// TIA Portal V17 export
// export: Created 2022-07-20T07:02:30.5184204Z, ExportSetting WithDefaults, DisplayName Totally Integrated Automation Portal, DisplayVersion V17, DisplayName TIA Portal Openness, DisplayVersion V17, DisplayName TIA Portal Version Control Interface, DisplayVersion V17, DisplayName SINAMICS Startdrive Advanced, DisplayVersion V17, DisplayName SINAMICS Startdrive G130, G150, S120, S150, SINAMICS MV, S210, DisplayVersion V17, DisplayName SINAMICS Startdrive G110M, G120, G120C, G120D, G120P, G115D, DisplayVersion V17, DisplayName STEP 7 Professional, DisplayVersion V17, DisplayName STEP 7 Safety, DisplayVersion V17, DisplayName WinCC Advanced, DisplayVersion V17
FUNCTION_BLOCK "FB11003_CamConvertProfile"   // FB11003, LAD
TITLE = Transfert and check data of foil profile
{ S7_Optimized_Access := 'TRUE' }
VERSION : 0.1
// stored: AutoNumber false, IsIECCheckEnabled false, IsRetainMemResEnabled false, MemoryReserve 100, SetENOAutomatically false, UDAEnableTagReadback false
   VAR_INPUT
      SheetProfile { ExternalAccessible := 'False'; ExternalVisible := 'False'; ExternalWritable := 'False'} : "stSheetProfile";
      FoilAcceleration : Real;
      FoilDeceleration : Real;
      RatioFoilPaper : Real := 1.0;
      CompensationForTensionInAcceleration : Real;
      CompensationForTensionInDeceleration : Real;
      MainDriveVelocity : Real;
      DistanceProductSensorFilmDrum : Real;
      Execute { ExternalAccessible := 'False'; ExternalVisible := 'False'; ExternalWritable := 'False'} : Bool;
   END_VAR
   VAR_OUTPUT
      Done { ExternalAccessible := 'False'; ExternalVisible := 'False'; ExternalWritable := 'False'} : Bool;
      Error { ExternalAccessible := 'False'; ExternalVisible := 'False'; ExternalWritable := 'False'} : Bool;
      DeadZoneBeforeStampArea { ExternalAccessible := 'False'; ExternalVisible := 'False'; ExternalWritable := 'False'} : Real;
      DeadZoneAfterStampArea { ExternalAccessible := 'False'; ExternalVisible := 'False'; ExternalWritable := 'False'} : Real;
      GapBetweenArea : Real;
      NbPoints : Real;
      CamProfile { ExternalAccessible := 'False'; ExternalVisible := 'False'; ExternalWritable := 'False'} : Array[1..32] of "LCamHdl_typeBasicPoint";
   END_VAR
   VAR
      statNumberOfArea : UInt;
      FoilAccelerationDistance : Real;   // [mm]
      FoilDecelerationDistance : Real;   // [mm]
      MasterAccelerationDistance : Real;
      MasterDecelerationDistance : Real;
      statPointtNumber { ExternalAccessible := 'False'; ExternalVisible := 'False'; ExternalWritable := 'False'} : UInt;
      statDone : Bool;
      statError : Bool;
      R_TRIG_Execute : R_TRIG;
   END_VAR
   VAR_TEMP
      AreaNumber : UInt;
      tempTotLength : Real;
   END_VAR
   VAR CONSTANT
      ratioDeadZone : Real := 4.0;
   END_VAR
   // // SheetProfile.Length : [mm]
BEGIN

REGION Network 1 (SCL): Comments
   //==========================================================================================
   // SIEMENS SAS      RC-FR DI FA APC
   //------------------------------------------------------------------------------------------
   // Restrictions:    TIA V16 and more
   // Requirements:    S7-1500T + LCameHdl + MGI library
   // Functionality:   This function block convert stSheetProfile into LCamHdl advanced element
   // and check data
   //------------------------------------------------------------------------------------------
   // Change log table:
   // Version      Date        Expert in charge    Changes applied
   // 01.00.01     09.06.2020  RTO                 First released version
   //==========================================================================================
END_REGION

REGION Network 2 (SCL): Edge Signals & Timers
   REGION EDGE SIGNALS
       #R_TRIG_Execute(CLK := #Execute);
   END_REGION
END_REGION

REGION Network 3 (SCL): Manage data
   IF NOT #Execute THEN
       #statDone := FALSE;
       #statError := FALSE;
   END_IF;

   IF #R_TRIG_Execute.Q THEN

       REGION Parameters
           // Get number of area used
           #statNumberOfArea := 0;
           FOR #AreaNumber := 1 TO "MAX_NUMBER_OF_FOIL_AREA" DO
               IF #SheetProfile.Area[#AreaNumber].Start <> #SheetProfile.Area[#AreaNumber].End THEN
                   #statNumberOfArea := #statNumberOfArea + 1;
               END_IF;
           END_FOR;

           // Get foil acceleration and deceleration distance
           #FoilAccelerationDistance := #FoilAcceleration * #ratioDeadZone;
           #FoilDecelerationDistance := #FoilDeceleration * #ratioDeadZone;

           // Get winder acceleration and deceleration distance

           #MasterAccelerationDistance := #FoilAccelerationDistance;// / #RatioFoilPaper;
           #MasterDecelerationDistance := #FoilDecelerationDistance;// / #RatioFoilPaper;

               // Parameters error
               IF #statNumberOfArea = 0
                   OR #FoilAccelerationDistance <= 0
                   OR #FoilDecelerationDistance <= 0
               THEN
                   #statError := TRUE;
               END_IF;

           // Clear CamProfile
           FOR #statPointtNumber := 1 TO 32 DO
               #CamProfile[#statPointtNumber].leadingValue := 0.0;
               #CamProfile[#statPointtNumber].followingValue := 0.0;
               #CamProfile[#statPointtNumber].velocityRatio := 0.0;
               #CamProfile[#statPointtNumber].accelerationRatio := 0.0;
           END_FOR;

           // Initializr number of segment
           #statPointtNumber := 1;

       END_REGION

       IF NOT #statError THEN
           REGION Segment definition
               //--- FIRST POINT ---
               #CamProfile[#statPointtNumber].leadingValue := - #DistanceProductSensorFilmDrum;
               #CamProfile[#statPointtNumber].followingValue := 0.0;
               #CamProfile[#statPointtNumber].velocityRatio := 0.0;
               #CamProfile[#statPointtNumber].accelerationRatio := 0.0;
               #statPointtNumber := #statPointtNumber + 1;

               //--- AREA ---
               FOR #AreaNumber := 1 TO #statNumberOfArea DO
                   //--- ACCELERATION ---
                   // From
                   #CamProfile[#statPointtNumber].leadingValue := #SheetProfile.Area[#AreaNumber].Start + #SheetProfile.StampAreaStartAdjustment - #MasterAccelerationDistance;//;#FoilAccelerationDistance;
                   #CamProfile[#statPointtNumber].followingValue := #CamProfile[#statPointtNumber-1].followingValue;
                   #CamProfile[#statPointtNumber].velocityRatio := 0.0;
                   #CamProfile[#statPointtNumber].accelerationRatio := 0.0;
                   #statPointtNumber := #statPointtNumber + 1;
                   // To
                   #CamProfile[#statPointtNumber].leadingValue := #SheetProfile.Area[#AreaNumber].Start + #SheetProfile.StampAreaStartAdjustment + #CompensationForTensionInAcceleration;
                   #CamProfile[#statPointtNumber].followingValue := #CamProfile[#statPointtNumber - 1].followingValue + #FoilAccelerationDistance + #CompensationForTensionInAcceleration;//#UnwinderAccelerationDistance + 15.0;
                   #CamProfile[#statPointtNumber].velocityRatio := #RatioFoilPaper;
                   #CamProfile[#statPointtNumber].accelerationRatio := 0.0;
                   #statPointtNumber := #statPointtNumber + 1;

                       // Error accemeration segment
                       IF #CamProfile[#statPointtNumber-1].leadingValue < #CamProfile[#statPointtNumber-2].leadingValue
                       OR #CamProfile[#statPointtNumber-1].followingValue < #CamProfile[#statPointtNumber-2].followingValue
                       THEN
                           #statError := TRUE;
                       END_IF;

                   //--- SYNCHRONOUS ---
                   // Until
                   #CamProfile[#statPointtNumber].leadingValue := #CamProfile[#statPointtNumber-1].leadingValue + #SheetProfile.Area[#AreaNumber].End - #SheetProfile.Area[#AreaNumber].Start + #SheetProfile.StampAreaLengthAdjustement;
                   #CamProfile[#statPointtNumber].followingValue := #CamProfile[#statPointtNumber - 1].followingValue + (#SheetProfile.Area[#AreaNumber].End - #SheetProfile.Area[#AreaNumber].Start) * #RatioFoilPaper + #SheetProfile.StampAreaLengthAdjustement;
                   #CamProfile[#statPointtNumber].velocityRatio := #RatioFoilPaper;
                   #CamProfile[#statPointtNumber].accelerationRatio := 0.0;
                   #statPointtNumber := #statPointtNumber + 1;


                       // Error synchronous segment
                   IF #CamProfile[#statPointtNumber - 1].leadingValue < #CamProfile[#statPointtNumber - 2].leadingValue
                       OR #CamProfile[#statPointtNumber - 1].followingValue < #CamProfile[#statPointtNumber - 2].followingValue
                   THEN
                       #statError := TRUE;
                   END_IF;

                   //--- DECELERATION ---
                   // Until
                   #CamProfile[#statPointtNumber].leadingValue := #CamProfile[#statPointtNumber - 1].leadingValue + #MasterDecelerationDistance + (#CompensationForTensionInDeceleration/1.0);//#FoilDecelerationDistance;
                       #CamProfile[#statPointtNumber].followingValue := #CamProfile[#statPointtNumber - 1].followingValue + #FoilDecelerationDistance + #CompensationForTensionInDeceleration;//#UnwinderDecelerationDistance + 10.0;
                   #CamProfile[#statPointtNumber].velocityRatio := 0.0;
                   #CamProfile[#statPointtNumber].accelerationRatio := 0.0;
                   #statPointtNumber := #statPointtNumber + 1;

                       // Error decelration segment
                       IF #CamProfile[#statPointtNumber - 1].leadingValue < #CamProfile[#statPointtNumber - 2].leadingValue
                       OR #CamProfile[#statPointtNumber - 1].followingValue < #CamProfile[#statPointtNumber - 2].followingValue
                       THEN
                           #statError := TRUE;
                       END_IF;

               END_FOR;
               //--- END AREA ---

               END_REGION
       END_IF;

       #statDone := TRUE;
   END_IF;
END_REGION

REGION Network 4 (SCL): Manage output
   REGION Output
       #DeadZoneBeforeStampArea := #FoilAcceleration * #ratioDeadZone;//#MasterAccelerationDistance;
       #DeadZoneAfterStampArea := #FoilDeceleration * #ratioDeadZone;//#MasterDecelerationDistance;
       #GapBetweenArea := #DeadZoneBeforeStampArea + #DeadZoneAfterStampArea;//#FoilAccelerationDistance + #FoilDecelerationDistance;
       #NbPoints := #statPointtNumber-1;
       #Done := #statDone;
       #Error := #statError;
   END_REGION
END_REGION
END_FUNCTION_BLOCK
